(* PLC project Tc2_Utilities.FB_LocalSystemTime Demo, tc3-libraries-kb TwinCAT 3.1 *)
(* stored: creationDateTime 2026-05-10T20:00:00, modificationDateTime 2026-05-10T20:00:00 *)

PROGRAM P_Demo_FB_LocalSystemTime
  VAR
    fbFB_LocalSystemTime : FB_LocalSystemTime;  (* Tc2_Utilities.FB_LocalSystemTime 实例 *)
    arg_sNetID : T_AmsNetID;  (* VAR_INPUT sNetID *)
    arg_bEnable : BOOL;  (* VAR_INPUT bEnable *)
    arg_dwCycle : DWORD(1..86400);  (* VAR_INPUT dwCycle *)
    arg_dwOpt : DWORD;  (* VAR_INPUT dwOpt *)
    arg_tTimeout : TIME;  (* VAR_INPUT tTimeout *)
    out_bValid : BOOL;  (* VAR_OUTPUT bValid *)
    out_systemTime : TIMESTRUCT;  (* VAR_OUTPUT systemTime *)
    out_tzID : E_TimeZoneID;  (* VAR_OUTPUT tzID *)
  END_VAR

            // ============================================================
// Tc2_Utilities.FB_LocalSystemTime 演示程序（FB 实例）
// ============================================================
// 验证步骤：
//   1. 引用 Tc2_Utilities（及依赖类型所在库 Tc2_System 等）
//   2. 编译 + 登录
//   3. 按 doc.md 给 arg_* 赋值
//   4. 在线监视 out_* / io_* 输出
// ============================================================

fbFB_LocalSystemTime(
    sNetID := arg_sNetID,
    bEnable := arg_bEnable,
    dwCycle := arg_dwCycle,
    dwOpt := arg_dwOpt,
    tTimeout := arg_tTimeout,
    bValid => out_bValid,
    systemTime => out_systemTime,
    tzID => out_tzID
);

          
END_PROGRAM
